ADAPTER INeredaAct (* Adapter Interface *)
  (* Standard: 61499-1 *)
  (* Version 0.0, 6/7/2026, Schneider Electric *)
  PACKAGE SE.Nereda;
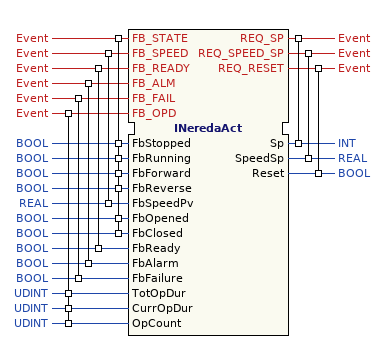
  EVENT_INPUT
    FB_STATE WITH FbStopped, FbRunning, FbForward, FbReverse, FbOpened, FbClosed;
    FB_SPEED WITH FbSpeedPv;
    FB_READY WITH FbReady;
    FB_ALM WITH FbAlarm;
    FB_FAIL WITH FbFailure;
    FB_OPD WITH TotOpDur, CurrOpDur, OpCount;
  END_EVENT
  EVENT_OUTPUT
    REQ_SP WITH Sp;
    REQ_SPEED_SP WITH SpeedSp;
    REQ_RESET WITH Reset;
  END_EVENT
  VAR_INPUT
    FbStopped : BOOL;
    FbRunning : BOOL;
    FbForward : BOOL;
    FbReverse : BOOL;
    FbSpeedPv : REAL;
    FbOpened : BOOL;
    FbClosed : BOOL;
    FbReady : BOOL;
    FbAlarm : BOOL;
    FbFailure : BOOL;
    TotOpDur : UDINT;
    CurrOpDur : UDINT;
    OpCount : UDINT;
  END_VAR
  VAR_OUTPUT
    Sp : INT;
    SpeedSp : REAL;
    Reset : BOOL;
  END_VAR
  SERVICE SOCKET/PLUG
    SEQUENCE request_confirm
      SOCKET.REQ(REQD) -> PLUG.REQ(REQD);
      PLUG.CNF(CNFD) -> SOCKET.CNF(CNFD);
    END_SEQUENCE
    SEQUENCE indication_response
      PLUG.IND(INDD) -> SOCKET.IND(INDD);
      SOCKET.RSP(RSPD) -> PLUG.RSP(RSPD);
    END_SEQUENCE
  END_SERVICE
END_ADAPTER
